FUNCTION_BLOCK ToggleRelaysWithDelay
VAR_INPUT
    StartDelayToggle : BOOL;           // Button from HMI
    DelayMsInput : INT;                // Delay in ms from HMI
END_VAR

VAR_IN_OUT
    BoolRelayArray : ARRAY[1..22] OF BOOL; // Relay control array
END_VAR

VAR
    Timer : TON;                       // Delay timer
    RelayIndex : INT := 1;             // Current relay index
    DelayTime : TIME;                  // Converted delay
    State : INT := 0;                  // 0: idle, 1: toggling on, 2: toggling off
    Latch : BOOL := FALSE;             // For edge detection
    MaxRelaysToggled : INT := 0;       // Keep track of how many relays were toggled ON
END_VAR


// Convert Delay input
DelayTime := INT_TO_TIME(DelayMsInput); //* 1ms;

// Detect rising/falling edge
IF StartDelayToggle AND NOT Latch THEN
    // Start toggle ON sequence
    State := 1;
    RelayIndex := 1;
    MaxRelaysToggled := 0;
    Timer(IN := FALSE);
ELSIF NOT StartDelayToggle AND Latch THEN
    // If toggle was ON but now turned OFF
    IF State = 1 THEN
        // Was toggling ON – cancel and reverse off relays
        State := 2;
        RelayIndex := RelayIndex - 1;
        IF RelayIndex < 1 THEN
            RelayIndex := 1;
        END_IF
    ELSIF State = 0 THEN
        // If already finished, now start toggling OFF
        State := 2;
        RelayIndex := 22;
    END_IF
END_IF
Latch := StartDelayToggle;

// Relay ON Sequence
IF State = 1 THEN
    Timer(IN := TRUE, PT := DelayTime);
    IF Timer.Q THEN
        BoolRelayArray[RelayIndex] := TRUE;
        MaxRelaysToggled := RelayIndex;
        RelayIndex := RelayIndex + 1;
        Timer(IN := FALSE); // Reset timer
        IF RelayIndex > 22 THEN
            State := 0; // Done
        END_IF
    END_IF

// Relay OFF Sequence (reverse)
ELSIF State = 2 THEN
    Timer(IN := TRUE, PT := DelayTime);
    IF Timer.Q THEN
        BoolRelayArray[RelayIndex] := FALSE;
        RelayIndex := RelayIndex - 1;
        Timer(IN := FALSE); // Reset timer
        IF RelayIndex < 1 THEN
            State := 0; // Done
        END_IF
    END_IF
END_IF

END_FUNCTION_BLOCK

(* stored: Version 1.1.0.1, ProductVersion 3.1.4024.13
   POU ToggleRelaysWithDelay: Id {672ec801-d5d4-4ea2-8f3a-4853371ff3c7}, SpecialFunc None *)
